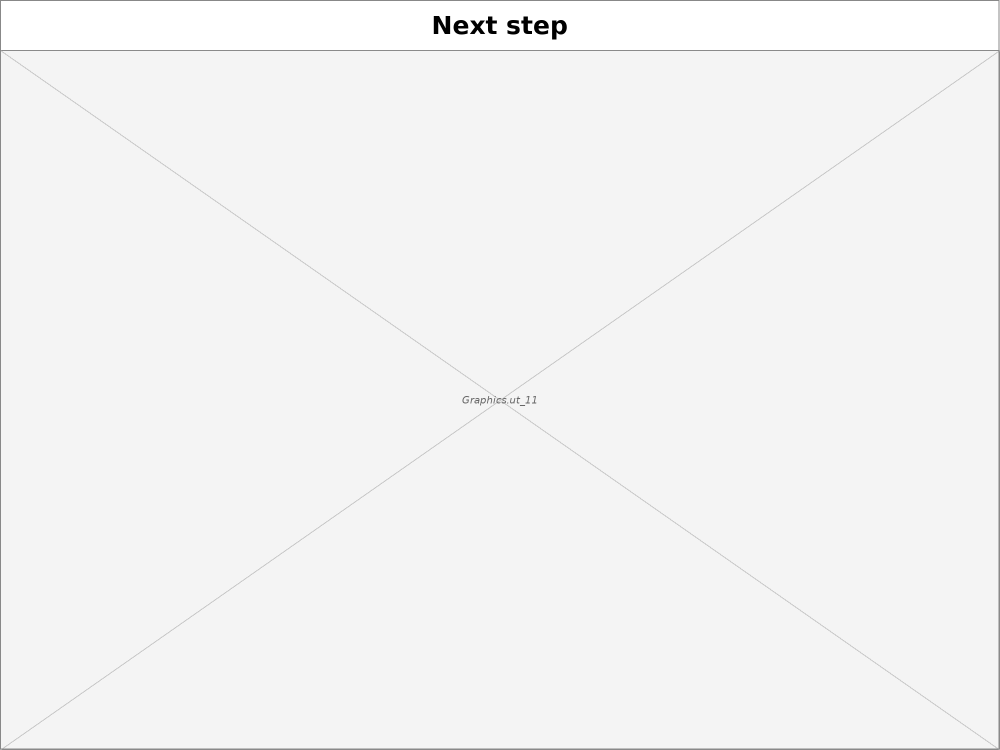
VISUALIZATION vTransporterSequence  // 1000x750
VAR_IN_OUT
	iWorkStep	: INT;
END_VAR
    Image (0,50 1000x700), invisible if: NOT( iWorkStep = 10 ), image: Graphics.ut_1
    Image (0,50 1000x700), invisible if: NOT( iWorkStep = 14 OR iWorkStep = 12), image: Graphics.ut_2
    Image (0,50 1000x700), invisible if: NOT( iWorkStep = 18 OR iWorkStep = 16), image: Graphics.ut_3
    Image (0,50 1000x700), invisible if: NOT( iWorkStep = 20), image: Graphics.ut_4
    Image (0,50 1000x700), invisible if: NOT( iWorkStep = 22), image: Graphics.ut_5
    Image (0,50 1000x700), invisible if: NOT (iWorkStep = 24 OR iWorkStep = 25), image: Graphics.ut_6
    Image (0,50 1000x700), invisible if: NOT (iWorkStep = 26), image: Graphics.ut_7
    Image (0,50 1000x700), invisible if: NOT( iWorkStep = 28), image: Graphics.ut_8
    Image (0,50 1000x700), invisible if: NOT( iWorkStep = 30), image: Graphics.ut_9
    Image (0,50 1000x700), invisible if: NOT( iWorkStep = 32), image: Graphics.ut_10
    Image (0,50 1000x700), invisible if: NOT( iWorkStep = 34), image: Graphics.ut_11
    Label (0,0 1000x50), "Next step"
END_VISUALIZATION

(* stored: Version 1.1.0.1, ProductVersion 3.1.4024.13
   Visu vTransporterSequence: Id {8eb95215-ccdf-4018-bdb0-fe3b41679847} *)
